FUNCTION_BLOCK FB_LightControl_OnOff implements I_LightControl
VAR_INPUT
END_VAR
VAR_OUTPUT
END_VAR
VAR
END_VAR

{warning 'add method implementation'}
METHOD M_Reset : BOOL
END_METHOD

{warning 'add method implementation'}
METHOD M_Set : BOOL
END_METHOD

{warning 'add property implementation'}
PROPERTY nAddress : DINT
GET
END_GET
SET
END_SET
END_PROPERTY

{warning 'add property implementation'}
PROPERTY nIlluminance : REAL
GET
END_GET
SET
END_SET
END_PROPERTY

END_FUNCTION_BLOCK

(* stored: Version 1.1.0.1, ProductVersion 3.1.4022.18
   POU FB_LightControl_OnOff: Id {f51cf791-f61e-4838-a54c-1845cb90087a}, SpecialFunc None
   Method M_Reset: Id {85ed67b8-9563-491f-90fe-00d72be67a2e}
   Method M_Set: Id {f42b4bf1-c525-44ed-8944-31a3b34c3d3d}
   Property nAddress: Id {d9ff440f-ac1e-4bf0-a984-91af453e2734}
   Get Get: Id {76706d52-e499-4a47-86d5-6bd5a7d4412b}
   Set Set: Id {98a3f403-31d3-49eb-b917-1c7eeebf72ba}
   Property nIlluminance: Id {8b1d9e45-1273-435f-a58a-88a965e23b67}
   Get Get: Id {67c9a7fa-2c37-433d-8ec7-7a51190057e6}
   Set Set: Id {2fae2e5e-8dae-445e-9603-b8edb0740b6a} *)
